// TIA Portal project "Project1" (V18)

(* hardware
DEVICE "S7-1200 station_1"  S7-1200 Station
   slot 0: "Rack_0"  S7-1200 Rack  Rack  V1.0
   slot 1: "PLC_1"  CPU 1214C AC/DC/Rly  6ES7 214-1BG40-0XB0  V4.1
   slot 2: "DI 16x24VDC_1"  6ES7 221-1BH32-0XB0  V2.0
   slot 101: "CM 1241 (RS232)_1"  6ES7 241-1AH30-0XB0  V1.0
*)

// ===== PLC "PLC_1"  CPU 1214C AC/DC/Rly =====

VAR_GLOBAL   // PLC tag table "Default tag table"
   "start_1" AT %I0.0 : Bool;
   "start_2" AT %I0.4 : Bool;
   "stop_1" AT %I0.1 : Bool;
   "stop_2" AT %I0.5 : Bool;
   "Proximity Sensor" AT %I0.3 : Bool;
   "Emergency button" AT %I0.2 : Bool;
   "PIR sensor" AT %I0.6 : Bool;
   "red light" AT %Q0.4 : Bool;
   "yellow light" AT %Q0.3 : Bool;
   "green light" AT %Q0.0 : Bool;
   "blue light" AT %Q0.2 : Bool;
   "white light" AT %Q0.1 : Bool;
   "led light" AT %Q0.5 : Bool;
   "Electro-valve" AT %Q0.6 : Bool;
   "Alarm_1" AT %Q0.7 : Bool;
   "Alarm_2" AT %Q1.0 : Bool;
END_VAR

DATA_BLOCK "inputs and outputs"   // DB1
{ S7_Optimized_Access := 'FALSE' }
VERSION : 0.1
   VAR
      inputs : Array[1..16] of Bool;
      outputs : Array[1..16] of Bool;
   END_VAR
BEGIN
END_DATA_BLOCK

ORGANIZATION_BLOCK "Main program"   // OB1, LAD, ProgramCycle
TITLE = "Main Program Sweep (Cycle)"
{ S7_Optimized_Access := 'TRUE' }
VERSION : 0.1
   VAR_INPUT
      Initial_Call : Bool;   // Initial call of this OB
      Remanence : Bool;   // =True, if remanent data are available
   END_VAR
BEGIN

REGION Network 1: latch and unlatch
   // using NO and NC contacts
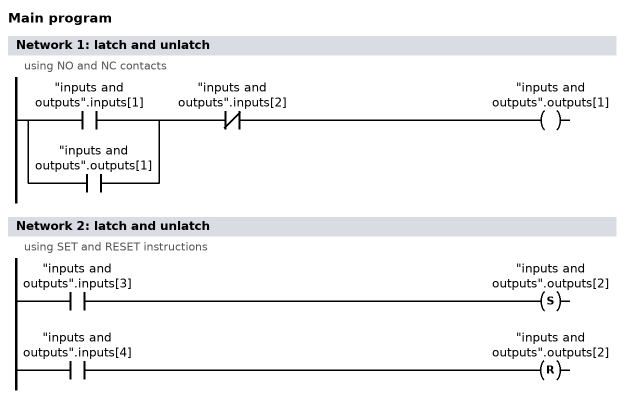
   RUNG wire#powerrail
      Contact( "inputs and outputs".inputs[1] )
      wire#w1
      I_Contact( "inputs and outputs".inputs[2] )
      Coil( "inputs and outputs".outputs[1] )
   END_RUNG
   RUNG wire#powerrail
      Contact( "inputs and outputs".outputs[1] )
   END_RUNG wire#w1
   // the same network as SCL:
   "inputs and outputs".outputs[1] := ("inputs and outputs".inputs[1] OR "inputs and outputs".outputs[1]) AND NOT "inputs and outputs".inputs[2];
END_REGION

REGION Network 2: latch and unlatch
   // using SET and RESET instructions
   RUNG wire#powerrail
      Contact( "inputs and outputs".inputs[3] )
      S_Coil( "inputs and outputs".outputs[2] )
   END_RUNG
   RUNG wire#powerrail
      Contact( "inputs and outputs".inputs[4] )
      R_Coil( "inputs and outputs".outputs[2] )
   END_RUNG
   // the same network as SCL:
   IF "inputs and outputs".inputs[3] THEN "inputs and outputs".outputs[2] := TRUE; END_IF;
   IF "inputs and outputs".inputs[4] THEN "inputs and outputs".outputs[2] := FALSE; END_IF;
END_REGION
END_ORGANIZATION_BLOCK